// Mitsubishi GX Works2 project: PLC_group31   PLC: FX3G

// global labels: Global1
VAR_GLOBAL
  DayStartSwitch AT X007 : BOOL;
  OngoingDayLamp AT Y007 : BOOL;
  WorkingDaySwitch AT X006 : BOOL;
  StorageSwitch AT X001 : BOOL;
  CreamInput AT D1110 : REAL;
  CreamAmount AT D1100 : REAL;
END_VAR
VAR_GLOBAL CONSTANT
  MinCream : REAL := 300;
END_VAR
VAR_GLOBAL
  CreamCheck AT M2 : BOOL;
  StartSwitch AT X007 : BOOL;
  ChocInput AT D1112 : REAL;
  ChockCheck AT M1 : BOOL;
  helpBulb AT M34 : BOOL;
  FlickerLamp1 AT M6 : BOOL;
END_VAR
VAR_GLOBAL CONSTANT
  ConstantFlicker_4 : INT := 4;
END_VAR
VAR_GLOBAL
  FlickerLamp2 AT M5 : BOOL;
  FlickerTimer1 AT TC0 : BOOL;
  Timer1_Value AT TS0 : BOOL;
  FlickerTimer2 AT TC1 : BOOL;
  Timer2_Value AT TS1 : BOOL;
  FlickerLampStop AT M4 : BOOL;
  Timer4 AT TC4 : BOOL;
END_VAR
VAR_GLOBAL CONSTANT
  TransTime : INT := 40;
END_VAR
VAR_GLOBAL
  StopFlicker AT TS4 : BOOL;
  FlickerTransfer1 AT Y000 : BOOL;
  FlickerTransfer2 AT Y001 : BOOL;
  TEST_helpBulb AT X000 : BOOL;
  Sample_Crust AT X006 : BOOL;
  BiscuitInput AT D1114 : REAL;
END_VAR
VAR_GLOBAL CONSTANT
  MinBisc : REAL := 6;
  MinChock : REAL := 240;
END_VAR
VAR_GLOBAL
  BiscCheck AT M3 : BOOL;
  CreamChock AT M2 : BOOL;
  Cream_inv AT D1100 : REAL;
  Chock_inv AT D1102 : REAL;
  Bisc_inv AT D1104 : REAL;
  Checcc AT M8 : BOOL;
  phase_1 AT X011 : BOOL;
END_VAR
VAR_GLOBAL CONSTANT
  sprinkling : REAL := 300;
END_VAR
VAR_GLOBAL
  cont_sprink AT D1106 : REAL;
  First_move AT M3 : BOOL;
END_VAR
VAR_GLOBAL CONSTANT
  const5 : REAL := 5;
  normalSize_Deep : REAL := 120;
END_VAR
VAR_GLOBAL
  cont_deep AT D1108 : REAL;
  DeepType AT M7 : BOOL;
  THISISWORKING AT X006 : BOOL;
  WORKINGTEST AT M9 : BOOL;
  analog_input1 AT D8280 : REAL;
  Save_analog AT D1116 : REAL;
END_VAR
VAR_GLOBAL CONSTANT
  DoubleSize_Deep : REAL := 240;
END_VAR
VAR_GLOBAL
  analog_input AT D8280 : INT;
  Save_analog1 AT D1116 : INT;
END_VAR
VAR_GLOBAL CONSTANT
  const_5 : INT := 5;
  Div_normAnalog : INT := 405;
END_VAR
VAR_GLOBAL
  machineB_timer AT TC3 : BOOL;
END_VAR
VAR_GLOBAL CONSTANT
  machineB_time : INT := 50;
END_VAR
VAR_GLOBAL
  stopMachineB AT TS3 : BOOL;
  machineB_lamp AT Y003 : BOOL;
  crembo_Package AT X000 : BOOL;
  first_five AT CC0 : BOOL;
  firstFive_lamp AT Y002 : BOOL;
  Out_firstFive AT CS0 : BOOL;
  last_crembo AT CC1 : BOOL;
END_VAR
VAR_GLOBAL CONSTANT
  const_6 : INT := 6;
END_VAR
VAR_GLOBAL
  Rest_cremboCounter AT Y002 : BOOL;
  Out_lastCrembo AT CS1 : BOOL;
  Cream_noLack AT M9 : BOOL;
  Bisc_noLack AT M10 : BOOL;
  Chock_noLack AT M11 : BOOL;
  Lack AT M8 : BOOL;
  Blink AT M10 : BOOL;
  startBlink_Enday AT M13 : BOOL;
  FlickeringTimer3 AT TC5 : BOOL;
END_VAR
VAR_GLOBAL CONSTANT
  Flicker2_Value : INT := 30;
END_VAR
VAR_GLOBAL
  FlickeringStoper3 AT TS5 : BOOL;
  Lac AT M8 : BOOL;
  finish_Package AT M14 : BOOL;
  start_day AT M15 : BOOL;
END_VAR
VAR_GLOBAL CONSTANT
  inital_cremboCounter : REAL;
  const6_crembos : REAL := 6;
END_VAR
VAR_GLOBAL
  output_cremboCounter AT D8282 : INT;
  crembo_Counter AT D1118 : REAL;
END_VAR
VAR_GLOBAL CONSTANT
  const40_normOutput : REAL := 40;
END_VAR
VAR_GLOBAL
  crembo_CounterINT AT D1120 : REAL;
  start_MachineA AT X010 : BOOL;
  MachineA_ON AT M0 : BOOL;
  stop_MachineA AT X005 : BOOL;
  sen_Touch AT X001 : BOOL;
  sen_Camera AT X002 : BOOL;
  sen_18 AT X003 : BOOL;
  sen_30 AT X004 : BOOL;
  sprink_sys AT Y004 : BOOL;
  sen_15 AT X003 : BOOL;
END_VAR
VAR_GLOBAL CONSTANT
  const0_empyCont : REAL;
END_VAR

// task Task_01 (event TRUE, interval 0, priority 31): POU_01

PROGRAM POU_01
(* structured ladder/FBD written out as ST: instructions are called as NAME(EN, inputs, outputs); _pN, _eN, _tN stand for wires *)
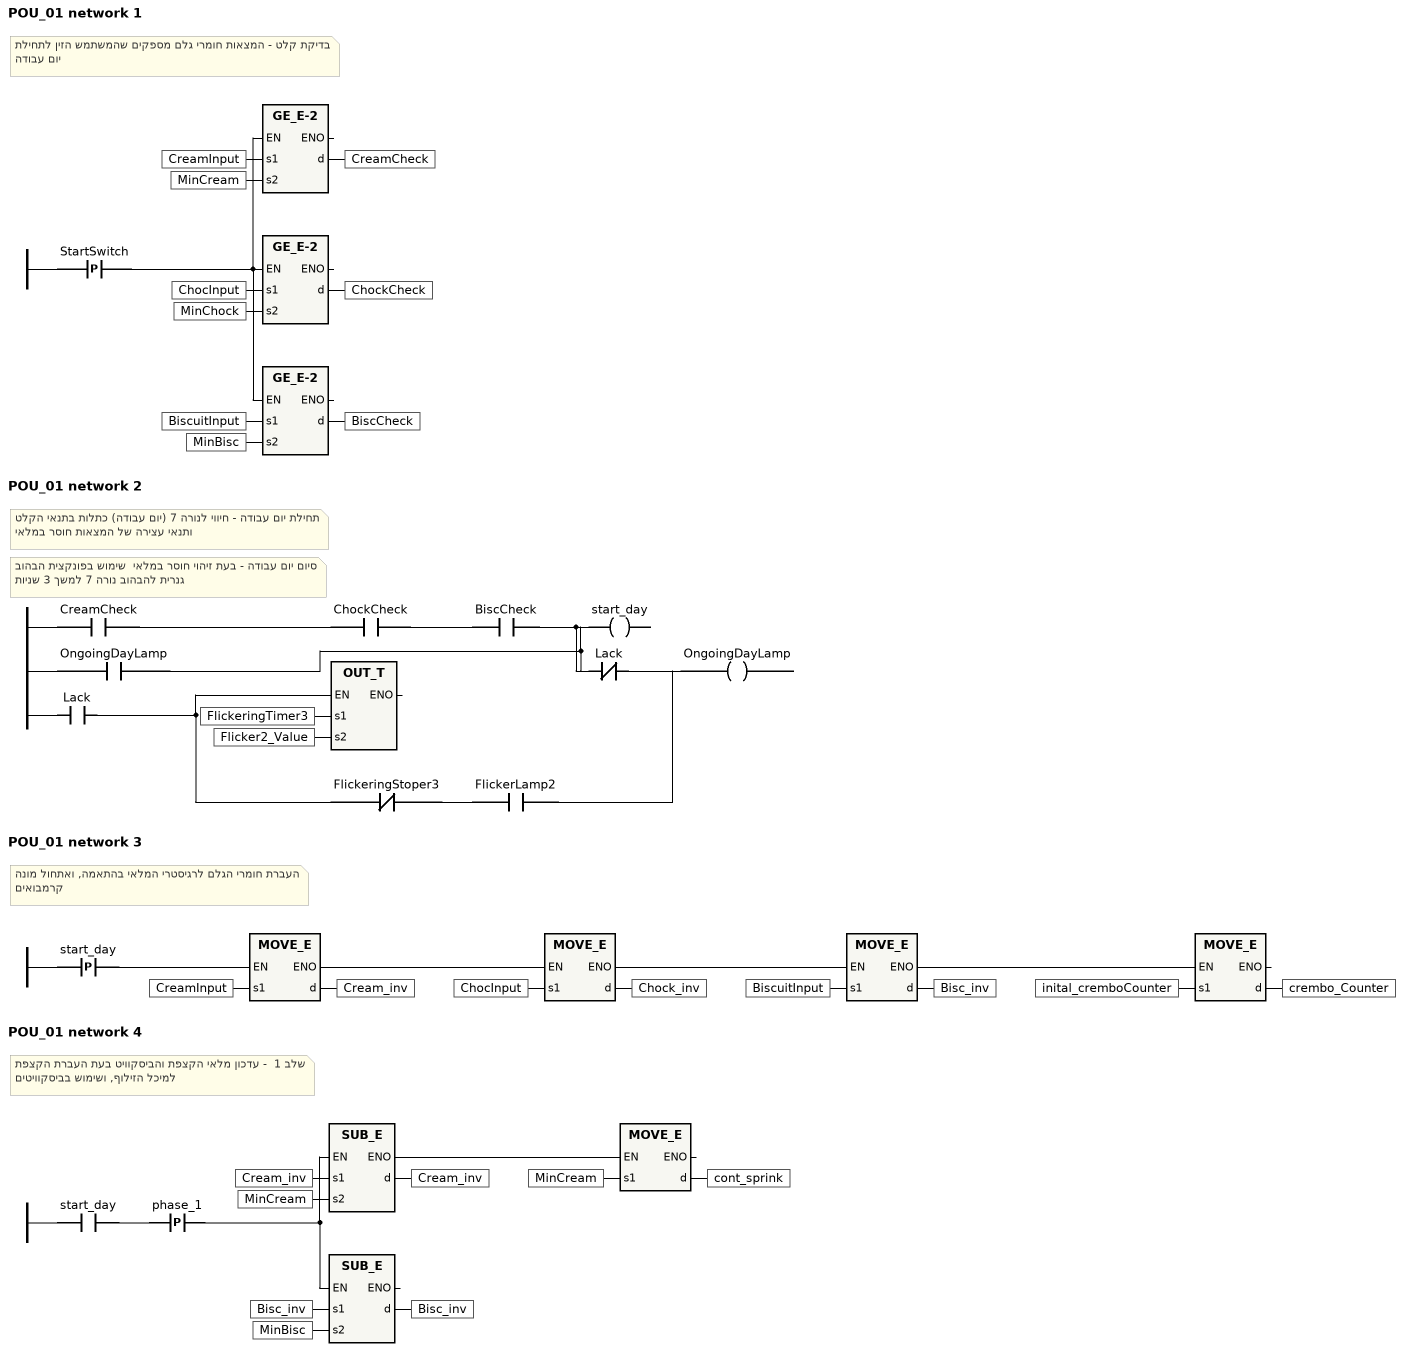
(* network 1 *)
(* בדיקת קלט - המצאות חומרי גלם מספקים שהמשתמש הזין לתחילת יום עבודה *)
_p1 := LDP(TRUE, StartSwitch);
GE_E(_p1, CreamInput, MinCream, CreamCheck);
GE_E(_p1, ChocInput, MinChock, ChockCheck);
GE_E(_p1, BiscuitInput, MinBisc, BiscCheck);
(* network 2 *)
(* תחילת יום עבודה - חיווי לנורה 7 (יום עבודה) כתלות בתנאי הקלט ותנאי עצירה של המצאות חוסר במלאי *)
(* סיום יום עבודה - בעת זיהוי חוסר במלאי  שימוש בפונקצית הבהוב גנרית להבהוב נורה 7 למשך 3 שניות *)
_p1 := (CreamCheck AND ChockCheck AND BiscCheck) OR OngoingDayLamp;
start_day := _p1;
OngoingDayLamp := (_p1 AND NOT Lack) OR (Lack AND NOT FlickeringStoper3 AND FlickerLamp2);
OUT_T(Lack, FlickeringTimer3, Flicker2_Value);
(* network 3 *)
(* העברת חומרי הגלם לרגיסטרי המלאי בהתאמה, ואתחול מונה קרמבואים *)
_e1 := MOVE_E(LDP(TRUE, start_day), CreamInput, Cream_inv);
_e2 := MOVE_E(_e1, ChocInput, Chock_inv);
_e3 := MOVE_E(_e2, BiscuitInput, Bisc_inv);
MOVE_E(_e3, inital_cremboCounter, crembo_Counter);
(* network 4 *)
(* שלב 1  - עדכון מלאי הקצפת והביסקוויט בעת העברת הקצפת למיכל הזילוף, ושימוש בביסקוויטים *)
_p1 := start_day AND LDP(TRUE, phase_1);
_e2 := SUB_E(_p1, Cream_inv, MinCream, Cream_inv);
MOVE_E(_e2, MinCream, cont_sprink);
SUB_E(_p1, Bisc_inv, MinBisc, Bisc_inv);
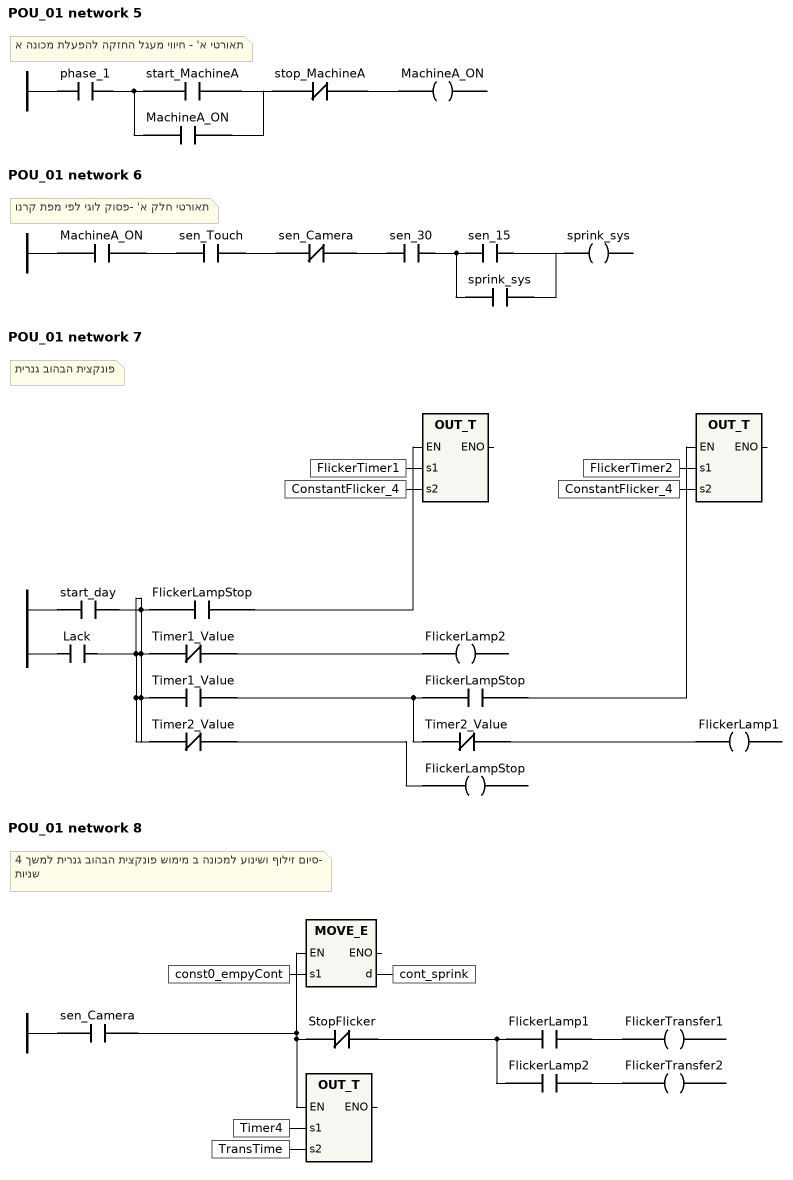
(* network 5 *)
(* תאורטי א' - חיווי מעגל החזקה להפעלת מכונה א *)
MachineA_ON := ((phase_1 AND start_MachineA) OR (phase_1 AND MachineA_ON)) AND NOT stop_MachineA;
(* network 6 *)
(* תאורטי חלק א' -פסוק לוגי לפי מפת קרנו *)
_p1 := MachineA_ON AND sen_Touch AND NOT sen_Camera AND sen_30;
sprink_sys := (_p1 AND sen_15) OR (_p1 AND sprink_sys);
(* network 7 *)
(* פונקצית הבהוב גנרית *)
_p1 := start_day OR Lack;
OUT_T(_p1 AND FlickerLampStop, FlickerTimer1, ConstantFlicker_4);
FlickerLamp2 := _p1 AND NOT Timer1_Value;
_p2 := _p1 AND Timer1_Value;
OUT_T(_p2 AND FlickerLampStop, FlickerTimer2, ConstantFlicker_4);
FlickerLamp1 := _p2 AND NOT Timer2_Value;
FlickerLampStop := _p1 AND NOT Timer2_Value;
(* network 8 *)
(* -סיום זילוף ושינוע למכונה ב מימוש פונקצית הבהוב גנרית למשך 4 שניות *)
MOVE_E(sen_Camera, const0_empyCont, cont_sprink);
_p1 := sen_Camera AND NOT StopFlicker;
FlickerTransfer1 := _p1 AND FlickerLamp1;
OUT_T(sen_Camera, Timer4, TransTime);
FlickerTransfer2 := _p1 AND FlickerLamp2;
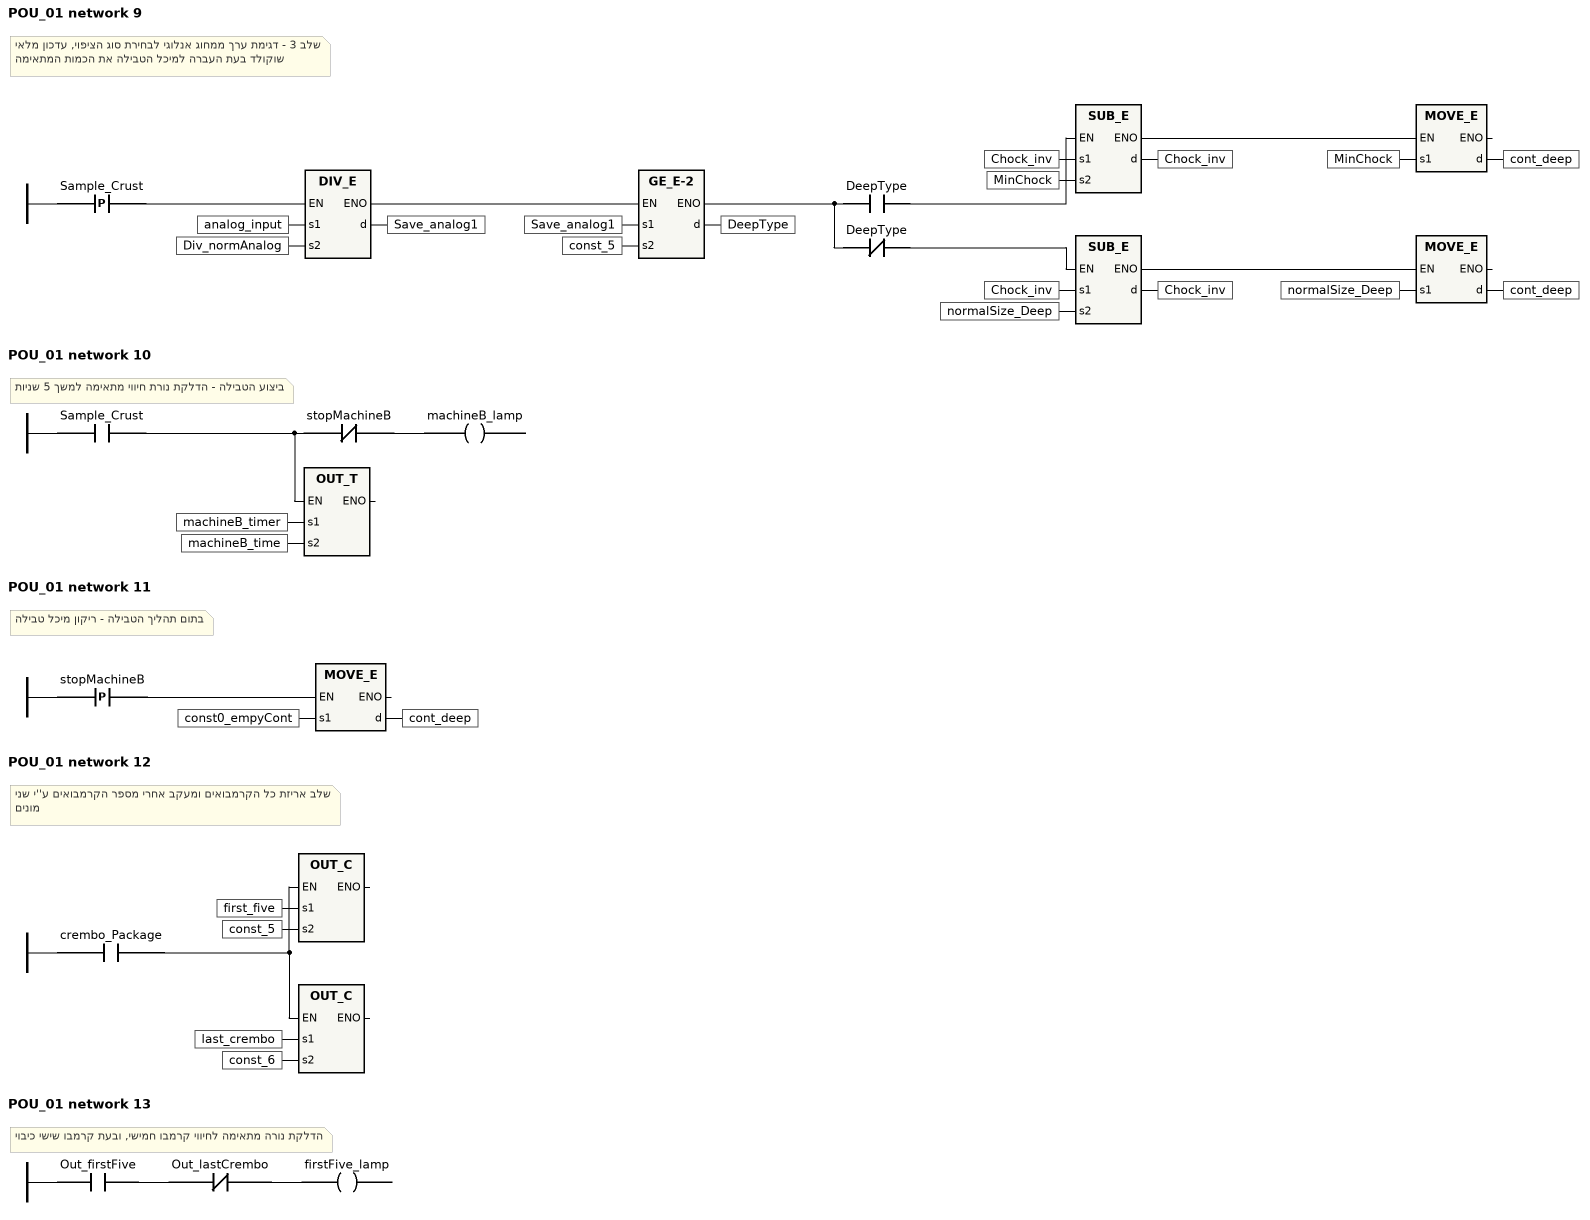
(* network 9 *)
(* שלב 3 - דגימת ערך ממחוג אנלוגי לבחירת סוג הציפוי, עדכון מלאי שוקולד בעת העברה למיכל הטבילה את הכמות המתאימה *)
_e1 := DIV_E(LDP(TRUE, Sample_Crust), analog_input, Div_normAnalog, Save_analog1);
_e2 := GE_E(_e1, Save_analog1, const_5, DeepType);
_e3 := SUB_E(_e2 AND DeepType, Chock_inv, MinChock, Chock_inv);
MOVE_E(_e3, MinChock, cont_deep);
_e4 := SUB_E(_e2 AND NOT DeepType, Chock_inv, normalSize_Deep, Chock_inv);
MOVE_E(_e4, normalSize_Deep, cont_deep);
(* network 10 *)
(* ביצוע הטבילה - הדלקת נורת חיווי מתאימה למשך 5 שניות *)
machineB_lamp := Sample_Crust AND NOT stopMachineB;
OUT_T(Sample_Crust, machineB_timer, machineB_time);
(* network 11 *)
(* בתום תהליך הטבילה - ריקון מיכל טבילה *)
MOVE_E(LDP(TRUE, stopMachineB), const0_empyCont, cont_deep);
(* network 12 *)
(* שלב אריזת כל הקרמבואים ומעקב אחרי מספר הקרמבואים ע''י שני מונים *)
OUT_C(crembo_Package, first_five, const_5);
OUT_C(crembo_Package, last_crembo, const_6);
(* network 13 *)
(* הדלקת נורה מתאימה לחיווי קרמבו חמישי, ובעת קרמבו שישי כיבוי *)
firstFive_lamp := Out_firstFive AND NOT Out_lastCrembo;
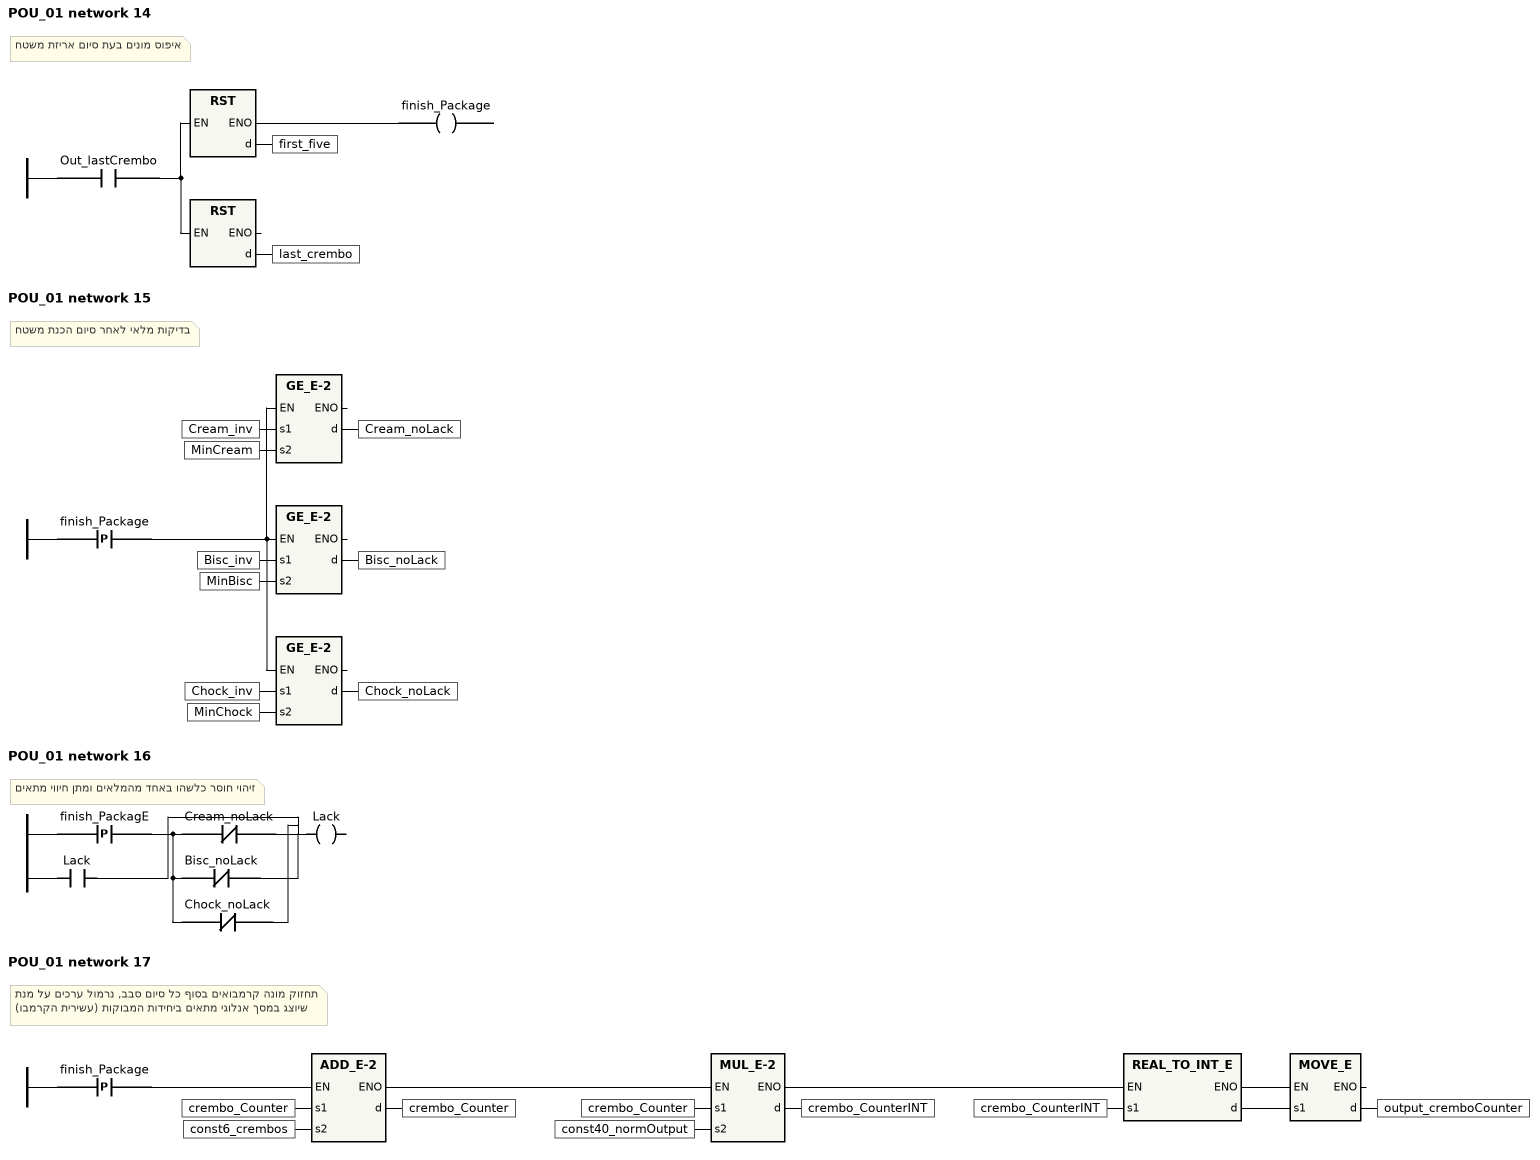
(* network 14 *)
(* איפוס מונים בעת סיום אריזת משטח *)
_e1 := RST(Out_lastCrembo, first_five);
finish_Package := _e1;
RST(Out_lastCrembo, last_crembo);
(* network 15 *)
(* בדיקות מלאי לאחר סיום הכנת משטח *)
_p1 := LDP(TRUE, finish_Package);
GE_E(_p1, Cream_inv, MinCream, Cream_noLack);
GE_E(_p1, Bisc_inv, MinBisc, Bisc_noLack);
GE_E(_p1, Chock_inv, MinChock, Chock_noLack);
(* network 16 *)
(* זיהוי חוסר כלשהו באחד מהמלאים ומתן חיווי מתאים *)
_p1 := LDP(TRUE, finish_PackagE);
Lack := (_p1 AND NOT Cream_noLack) OR (_p1 AND NOT Bisc_noLack) OR (_p1 AND NOT Chock_noLack) OR Lack;
(* network 17 *)
(* תחזוק מונה קרמבואים בסוף כל סיום סבב, נרמול ערכים על מנת שיוצג במסך אנלוגי מתאים ביחידות המבוקות (עשירית הקרמבו) *)
_e1 := ADD_E(LDP(TRUE, finish_Package), crembo_Counter, const6_crembos, crembo_Counter);
_e2 := MUL_E(_e1, crembo_Counter, const40_normOutput, crembo_CounterINT);
_e4 := REAL_TO_INT_E(_e2, crembo_CounterINT, _t3);
MOVE_E(_e4, _t3, output_cremboCounter);
END_PROGRAM
